///EL2502 | 2-channel pulse width output terminal 24 V DC
FUNCTION_BLOCK EL2502_v0_00

END_FUNCTION_BLOCK

(* stored: Version 1.1.0.1, ProductVersion 3.1.0.25
   POU EL2502_v0_00: Id {bdbebb5e-656b-423d-b816-7055e429268d} *)
